FUNCTION_BLOCK RandomEventConverter (* Basic Function Block Type *)
  (* Standard: 61499-2 *)
  (* Version 0.0, 8/30/2016, Dmitry, nxtControl GmbH, Template *)
  PACKAGE Main;
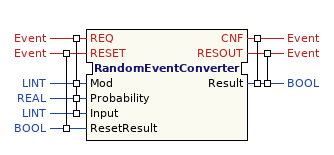
  EVENT_INPUT
    REQ WITH Mod, Probability, Input; (* Normal Execution Request *)
    RESET WITH ResetResult;
  END_EVENT
  EVENT_OUTPUT
    CNF WITH Result; (* Execution Confirmation *)
    RESOUT WITH Result;
  END_EVENT
  VAR_INPUT
    Mod : LINT;
    Probability : REAL;
    Input : LINT;
    ResetResult : BOOL;
  END_VAR
  VAR_OUTPUT
    Result : BOOL;
  END_VAR
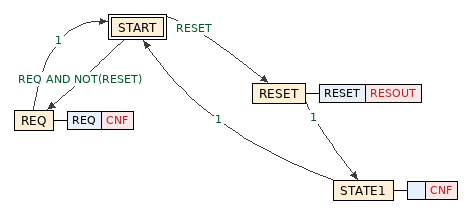
  EC_STATES
    START; (* Initial State *)
    REQ : REQ -> CNF; (* Normal execution *)
    RESET : RESET -> RESOUT;
    STATE1 : -> CNF;
  END_STATES
  EC_TRANSITIONS
    START TO REQ := REQ AND NOT(RESET);
    REQ TO START := 1;
    START TO RESET := RESET;
    RESET TO STATE1 := 1;
    STATE1 TO START := 1;
  END_TRANSITIONS
  ALGORITHM INIT IN ST: (* Initialization algorithm *)
;
  END_ALGORITHM
  ALGORITHM REQ IN ST: (* Normally executed algorithm *)
Result := (Mod - 1) * Probability >= ABS(Input MOD Mod);
  END_ALGORITHM
  ALGORITHM RESET IN ST:
Result := ResetResult;
  END_ALGORITHM
END_FUNCTION_BLOCK
